# EPICS autosave request: edgeApp/Db/NDEdge_settings.req
file "NDPluginBase_settings.req", P=$(P), R=$(R)
$(P)$(R)LowThreshold
$(P)$(R)ThresholdRatio
